# EPICS autosave request: measCompApp/Db/measCompUSBTempConfig_settings.req
$(P)$(R)TemperatureSensor
$(P)$(R)TemperatureWiring
